FUNCTION System : REFERENCE TO SystemBundle
VAR_INPUT
END_VAR
VAR
	bundle		: SystemBundle;
END_VAR


bundle.Call();

System REF= bundle;

END_FUNCTION

(* stored: Version 1.1.0.1, ProductVersion 3.1.4024.12
   POU System: Id {fd898ed2-9c53-4969-9e3a-245cd851a3ca}, SpecialFunc None *)
